FUNCTION_BLOCK FB_PumpGrundfosMagna3 EXTENDS FB_ActorContinous
VAR_INPUT
	nControlModeAutomatic : E_GrundfosMagna3ControlMode;
END_VAR
VAR_OUTPUT
END_VAR
VAR
	{attribute 'OPC.UA.DA' := '1'}
	localSetParameters : ST_PumpGrundfosMagna3SetParameters;
	{attribute 'OPC.UA.DA' := '1'}
	localState : ST_PumpGrundfosMagna3State;
	
	//I/O links
	//Inputs
	fTemperatureInternal_IN 	AT %I* : REAL; //°C
	fTemperatureExternal_IN 	AT %I* : REAL; //°C external temperature from sensor connected to pump
	fTemperatureDifference_IN	AT %I* : REAL; //°C
	fVolumeFlowRate_IN 			AT %I* : REAL; //m^3/h volume flow rate from pump
	fPressureDifference_IN	 	AT %I* : REAL; //pa = 10^-5 bar
	fPowerElectric_IN			AT %I* : REAL; //W
	fPowerThermal_IN	 		AT %I* : REAL; //W
	fRotationalSpeed_IN	 		AT %I* : REAL; //rpm
	fActualSetpoint_IN			AT %I* : REAL; //%
	bStatusOn_IN				AT %I* : BOOL; //True if pump is running
	nControlMode_IN				AT %I* : INT;	
	bAlarm_IN					AT %I* : BOOL; //True if pump has been stopped because of an alarm
	bWarning_IN					AT %I* : BOOL; //True if pump shows a warning
	bRemoteControlOn_IN			AT %I* : BOOL; //True if remote control is used
	nAlarmCode_IN				AT %I* : INT;
	nWarningCode_IN				AT %I* : INT;
	
	//Outputs
	bSetStatus_OUT 		AT %Q* : BOOL;	
	nControlMode_OUT	AT %Q* : INT;
	fSetPoint_OUT		AT %Q* : REAL;
	
	//internal variables:
	nControlMode : E_GrundfosMagna3ControlMode; //actual pump control mode
	bExternalTemperatureSensorConnected : BOOL := TRUE; //true if external temperature sensor connected
END_VAR

MAIN();
CalculateHydraulicPower();
SelectPumpControlMode();
SetState();

PROPERTY bExternalTemperatureSensor : BOOL
SET
bExternalTemperatureSensorConnected := bExternalTemperatureSensor;
END_SET
END_PROPERTY

METHOD CalculateHydraulicPower : REAL
VAR_INPUT
END_VAR
localState.fPowerHydraulic := localState.fPressureDifference*localState.fVolumeFlowRate;
END_METHOD

METHOD PROTECTED SelectPumpControlMode : BOOL
VAR_INPUT
END_VAR
IF control.bManualModeActivated THEN
	nControlMode := localSetParameters.nControlModeManual;
ELSIF control.bAlgorithmModeActivated AND algorithmPermission THEN
	nControlMode := localSetParameters.nControlModeAlgorithm;
ELSE
	nControlMode := nControlModeAutomatic;
END_IF
END_METHOD

METHOD PROTECTED   SetState : BOOL
VAR_INPUT
END_VAR
//Control state
controlState.bStatusOn := bStatusOn_IN;

//Error state
errorState.bError := bAlarm_IN;
errorState.bWarning := bWarning_IN;
errorState.sErrorMessage := CONCAT('Alarm code: ',INT_TO_STRING(nAlarmCode_IN));
errorState.sWarningMessage := CONCAT('Warning code: ',INT_TO_STRING(nWarningCode_IN));

//SetPoint state
setPointState.fOperatingPoint := fActualSetpoint_IN;
setPointState.fSetPoint := fSetPoint;

//Local state
localState.bRemoteControlOn := bRemoteControlOn_IN;
localState.fVolumeFlowRate := fVolumeFlowRate_IN;
localState.fTemperatureInternal := fTemperatureInternal_IN;
localState.fPressureDifference := fPressureDifference_IN;
localState.fPowerElectric := fPowerElectric_IN;
localState.fPowerThermal := fPowerThermal_IN;
localState.fRotationalSpeed := fRotationalSpeed_IN;

//Set external temperature and temperature difference if temperature sensor is connected
IF bExternalTemperatureSensorConnected THEN
	localState.fTemperatureExternal := fTemperatureExternal_IN;
	localState.fTemperatureDifference := fTemperatureDifference_IN;
END_IF;

//I/O-Links
nControlMode_OUT := nControlMode;
bSetStatus_OUT := bSetStatusOn;
fSetPoint_OUT := fSetPoint*100;
nControlMode_OUT := nControlMode;
END_METHOD

END_FUNCTION_BLOCK

(* stored: Version 1.1.0.1, ProductVersion 3.1.4024.9
   POU FB_PumpGrundfosMagna3: Id {5ff4732a-f57a-4b28-83eb-fee6b9ba074e}, SpecialFunc None
   Property bExternalTemperatureSensor: Id {61a8bc23-912e-42b7-8bba-85a22513c812}
   Set Set: Id {8af04288-c858-4540-ba92-3eea6e4d8f1e}
   Method CalculateHydraulicPower: Id {5ee59af5-7c08-4f03-8cfe-829337b66dfd}
   Method SelectPumpControlMode: Id {9f36f1dc-61c9-4f36-814e-95f20eaaf659}
   Method SetState: Id {ab5b0484-c37f-40fd-90a0-eb40d6c4211b} *)
